FUNCTION Convert_REAL_TO_REAL : Hresult
VAR_INPUT
	in : REAL;
	out : REFERENCE TO REAL;
END_VAR

out := in;

END_FUNCTION

(* stored: Version 1.1.0.1, ProductVersion 3.1.4024.12
   POU Convert_REAL_TO_REAL: Id {7ac5fd4e-0228-4550-918e-c1d9a60673d8}, SpecialFunc None *)
